{attribute 'qualified_only'}
{attribute 'strict'}

//Emuneration is a nickname given to integer value
TYPE myGenderType :
(
	unknown:=0,
	male,
	female
);
END_TYPE

(* stored: Version 1.1.0.1, ProductVersion 3.1.4024.11
   DUT myGenderType: Id {69621700-7f86-4eeb-8ae6-be1360454fdc} *)
